TYPE T_LongSTRING : STRING(1023);
END_TYPE

(* stored: Version 1.1.0.1
   DUT T_LongSTRING: Id {aec1c44f-8e00-4273-8791-bc4b03f1e76d} *)
